PROGRAM MAIN
VAR

	
	FCV_1: INT;
	FCV_2: INT;
	HopperLevel: REAL;
END_VAR

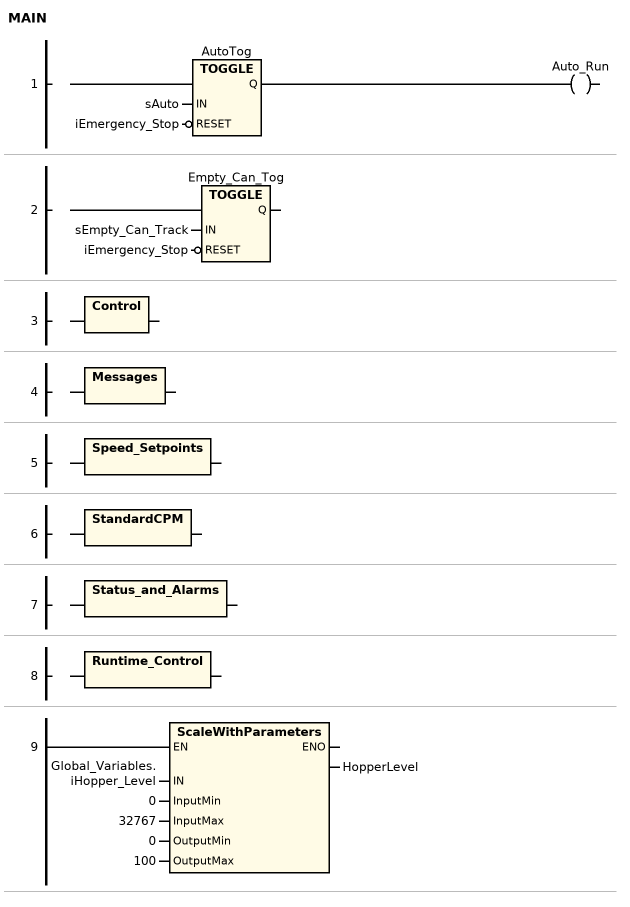
// NETWORK 1
AutoTog(IN := sAuto, RESET := NOT iEmergency_Stop); // TOGGLE
Auto_Run := AutoTog.Q;

// NETWORK 2
Empty_Can_Tog(IN := sEmpty_Can_Track, RESET := NOT iEmergency_Stop); // TOGGLE

// NETWORK 3
Control();

// NETWORK 4
Messages();

// NETWORK 5
Speed_Setpoints();

// NETWORK 6
StandardCPM();

// NETWORK 7
Status_and_Alarms();

// NETWORK 8
Runtime_Control();

// NETWORK 9
HopperLevel := ScaleWithParameters(IN := Global_Variables.iHopper_Level, InputMin := 0, InputMax := 32767, OutputMin := 0, OutputMax := 100);

END_PROGRAM

(* stored: Version 1.1.0.1, ProductVersion 3.1.4024.15
   POU MAIN: Id {c88d5593-508c-4327-a116-835b19cab405}, SpecialFunc None *)
